# B&R Automation Studio project DevProj
Automation Studio 4.10.2.37; technology packages: mappMotion 5.12.3

## Configuration Config1

CPU 5APC2200.AL14-000, AutomationRuntime B4.91, Build 4.1.2, Safety 0.0, Vc V4.72.3

### Task classes (Cpu.sw)
```
Cyclic#1:
  Main <- Programs.Main.prg
Binaries: udbdef, FWRules, TCData, sysconf, Role, User, iomap, ashwd, asfw, arconfig, ashwac
Libraries: standard, operator, runtime, astime, AsIecCon, Util, McBase, MpAxis, McAxis, MpBase, McAcpAx, PTP
```

### Hardware
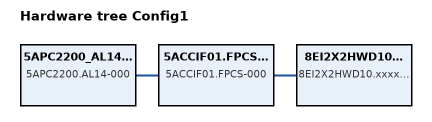
```
5ACCIF01.FPCS-000 : 5ACCIF01.FPCS-000 v1.8.1.0  [SL -> 5APC2200_AL14_000.SL1]
  Connector IF1:
    DNAConfiguration = manual
5APC2200_AL14_000 : 5APC2200.AL14-000 v2.0.1.0
  Connector IF3:
    AssignedOperatingSystem = ARemb
    ActivateDevice = 1
  Connector IF4:
    AssignedOperatingSystem = ARemb
    ActivateDevice = 1
  Connector IF5:
    AssignedOperatingSystem = ARemb
  Connector IF6:
    AssignedOperatingSystem = ARemb
  ConfigurationID = DevProj_Config1
  UserPartitionSize = 0
  TimerDeviceType = EPLX2X
  TimerDevice = 5ACCIF01.FPCS-000.IF1
  TaskClassIdleTime = 2000
  Cyclic1Tolerance = 0
  Cyclic2Duration = 10000
  Cyclic2Tolerance = 10000
  FileDevice1
  FileDeviceName1 = CNC_PrgDir
  FileDevicePath1 = C:\scUserFiles\
  ActivateOpcUa = 1
  OpcUa_AuthenticationSecurityPolicy_EnableNone = 1
  OpcUa_AuthenticationSecurityPolicy_EnableBasic128Rsa15 = 1
  OpcUa_Security_AdminRole = Everyone
  OpcUaLimitsMaxSessions = 4
  OpcUa_SamplingTimer_Default = 4
  OpcUaInformationModels_PV_Version = 1
8EI2X2HWD10.xxxx-1 : 8EI2X2HWD10.xxxx-1 v2.3.1.1  [PLK1 -> 5ACCIF01.FPCS-000.IF1 [Cable Type=PowerlinkCable, Length=10, Version=1.0.0.3]]
  DriveConfiguration/Module:
    McAcoposTypeID = AcoposP3DConfig
    ActivateACOPOSSimulationOnPLC = 1
  DriveConfiguration/Channel[1]/RealAxis:
    AxisReference = AxisX1_Link
  DriveConfiguration/Channel[1]/RealAxis/MechanicalElements/Gearbox:
    InputIsReadOnly = 0
    Input = 1
    OutputIsReadOnly = 0
    Output = 1
  DriveConfiguration/Channel[1]/RealAxis/MechanicalElements/RotaryToLinearTransformation:
    ReferenceDistanceIsReadOnly = 0
    ReferenceDistance = 1
  DriveConfiguration/Channel[1]/RealAxis/Controller:
    ModeIsReadOnly = 0
    Mode = PositionController
  DriveConfiguration/Channel[1]/RealAxis/Controller/Mode/Position:
    ProportionalGain = 50.0
    IntegrationTime = 0.0
    PredictionTime = 0.0004
    TotalDelayTime = 0.0004
  DriveConfiguration/Channel[1]/RealAxis/Controller/Mode/Speed:
    ProportionalGainIsReadOnly = 0
    ProportionalGain = 2.0
    IntegrationTimeIsReadOnly = 0
    IntegrationTime = 0.0
    FilterTimeIsReadOnly = 0
    FilterTime = 0.0
  DriveConfiguration/Channel[1]/RealAxis/Controller/Mode/LoopFilters:
    LoopFilter1 = NotUsed
    LoopFilter2 = NotUsed
    LoopFilter3 = NotUsed
  DriveConfiguration/Channel[1]/RealAxis/Homing:
    Mode = Direct
  DriveConfiguration/Channel[1]/RealAxis/Homing/Mode:
    Position = 0.0
    ReferencePulse = NotUsed
  DriveConfiguration/Channel[1]/RealAxis/Homing:
    RestorePositionVariable = 
  DriveConfiguration/Channel[1]/RealAxis/StopReaction:
    Quickstop = DecelerationLimit
    DriveError = DecelerationLimit
  DriveConfiguration/Channel[1]/RealAxis/MovementErrorLimits:
    PositionError = 1.0
    VelocityErrorMonitoring = Automatic1
  DriveConfiguration/Channel[1]/RealAxis:
    JerkFilter = NotUsed
  DriveConfiguration/Channel[1]/RealAxis/DigitalInputs/HomingSwitch:
    Source = NotUsed
    Level = High
  DriveConfiguration/Channel[1]/RealAxis/DigitalInputs/PositiveLimitSwitch:
    Source = NotUsed
    Level = High
  DriveConfiguration/Channel[1]/RealAxis/DigitalInputs/NegativeLimitSwitch:
    Source = NotUsed
    Level = High
  DriveConfiguration/Channel[1]/RealAxis/DigitalInputs/Trigger1:
    Source = X8Trigger1
    Level = High
  DriveConfiguration/Channel[1]/RealAxis/DigitalInputs/Trigger2:
    Source = X8Trigger2
    Level = High
  DriveConfiguration/Channel[1]/RealAxis/DigitalInputs/Quickstop:
    Input = Trigger2
  DriveConfiguration/Channel[1]/RealAxis/Simulation:
    SimulationModeOnPLC = SetValueGeneration
    SimulationModeOnACOPOS = NotUsed
  DriveConfiguration/Channel[2]/RealAxis:
    AxisReference = AxisZ1_Link
  DriveConfiguration/Channel[2]/RealAxis/MechanicalElements/Gearbox:
    InputIsReadOnly = 0
    Input = 1
    OutputIsReadOnly = 0
    Output = 1
  DriveConfiguration/Channel[2]/RealAxis/MechanicalElements/RotaryToLinearTransformation:
    ReferenceDistanceIsReadOnly = 0
    ReferenceDistance = 1
  DriveConfiguration/Channel[2]/RealAxis/Controller:
    ModeIsReadOnly = 0
    Mode = PositionController
  DriveConfiguration/Channel[2]/RealAxis/Controller/Mode/Position:
    ProportionalGain = 50.0
    IntegrationTime = 0.0
    PredictionTime = 0.0004
    TotalDelayTime = 0.0004
  DriveConfiguration/Channel[2]/RealAxis/Controller/Mode/Speed:
    ProportionalGainIsReadOnly = 0
    ProportionalGain = 2.0
    IntegrationTimeIsReadOnly = 0
    IntegrationTime = 0.0
    FilterTimeIsReadOnly = 0
    FilterTime = 0.0
  DriveConfiguration/Channel[2]/RealAxis/Controller/Mode/LoopFilters:
    LoopFilter1 = NotUsed
    LoopFilter2 = NotUsed
    LoopFilter3 = NotUsed
  DriveConfiguration/Channel[2]/RealAxis/Homing:
    Mode = Direct
  DriveConfiguration/Channel[2]/RealAxis/Homing/Mode:
    Position = 0.0
    ReferencePulse = NotUsed
  DriveConfiguration/Channel[2]/RealAxis/Homing:
    RestorePositionVariable = 
  DriveConfiguration/Channel[2]/RealAxis/StopReaction:
    Quickstop = DecelerationLimit
    DriveError = DecelerationLimit
  DriveConfiguration/Channel[2]/RealAxis/MovementErrorLimits:
    PositionError = 1.0
    VelocityErrorMonitoring = Automatic1
  DriveConfiguration/Channel[2]/RealAxis:
    JerkFilter = NotUsed
  DriveConfiguration/Channel[2]/RealAxis/DigitalInputs/HomingSwitch:
    Source = NotUsed
    Level = High
  DriveConfiguration/Channel[2]/RealAxis/DigitalInputs/PositiveLimitSwitch:
    Source = NotUsed
    Level = High
  DriveConfiguration/Channel[2]/RealAxis/DigitalInputs/NegativeLimitSwitch:
    Source = NotUsed
    Level = High
  DriveConfiguration/Channel[2]/RealAxis/DigitalInputs/Trigger1:
    Source = X8Trigger1
    Level = High
  DriveConfiguration/Channel[2]/RealAxis/DigitalInputs/Trigger2:
    Source = X8Trigger2
    Level = High
  DriveConfiguration/Channel[2]/RealAxis/DigitalInputs/Quickstop:
    Input = Trigger2
  DriveConfiguration/Channel[2]/RealAxis/Simulation:
    SimulationModeOnPLC = SetValueGeneration
    SimulationModeOnACOPOS = NotUsed
```

### ConfAxFea.axesgroupfeature - 5APC2200_AL14_000/mappMotion/ConfAxFea.axesgroupfeature
```
Element Feature_Programs (Type=axesgroupfeature)
  Type = Program
    ModalDataBehaviour = UseAxesGroupSettings
    InitialSettings:
      InterpolationTypes = LinearRapid
      PositionCoordinates = Absolute
      CircleCoordinates = Relative
      JACS_ACSProgramming = JACS
      ContourConnection = Inactive
      ProgrammingUnits = UseAxesGroupSettings
      Feedrates:
        FeedPath = Standard
        FeedCharacteristic = StandardCharacteristic
        FeedType = Feedrate
        FeedReduction = Inactive
        FeedrateValue = 0.0
        InverseFeedrateValue = 0.0
        FeedratePerRevValue = 0.0
    DefaultLanguage = BRGCode
    Location = Default
      FileDevice = CNC_PrgDir
    ProgramElements:
      PVs:
        PV[1]:
          PvName = ::RParams[31]
          Advanced:
            Alias = R31
            Synchronization = Ip
            Reference = No
Element Feature_Jogging (Type=axesgroupfeature)
  Type = Jogging
Element Feature_MFunctions (Type=axesgroupfeature)
  Type = MFunctions
    ModalDataBehaviour = UseAxesGroupSettings
    MFunction[1]:
      IndexType = Single
        Index = 31
      Blocking = Disabled
      Output = Before
      InSimulation = NotUsed
      PvMapping = ::M31
      Counter
```

### ConfAxes.axis - 5APC2200_AL14_000/mappMotion/ConfAxes.axis
```
Element AxisX1_Link (Type=axis)
  BaseTypeIsReadOnly = 0
  BaseType = LinearBounded
    MeasurementUnit = 5066068
    MeasurementResolutionIsReadOnly = 0
    MeasurementResolution = 0.01
    CountDirectionIsReadOnly = 0
    CountDirection = Standard
  MovementLimitsIsReadOnly = 0
  MovementLimits = Internal
    Position:
      LowerLimitMin = -1.79769313486231E308
      UpperLimitMax = 1.79769313486231E308
      LowerLimit = -1000.0
      UpperLimit = 1000.0
    VelocityIsReadOnly = 0
    Velocity:
      VelocityMax = 3.4E38
      Velocity = 10.0
    AccelerationIsReadOnly = 0
    Acceleration:
      AccelerationMax = 3.4E38
      Acceleration = 50.0
    DecelerationIsReadOnly = 0
    Deceleration:
      DecelerationMax = 3.4E38
      Deceleration = 50.0
  Alarms = None
Element AxisZ1_Link (Type=axis)
  BaseTypeIsReadOnly = 0
  BaseType = LinearBounded
    MeasurementUnit = 5066068
    MeasurementResolutionIsReadOnly = 0
    MeasurementResolution = 0.01
    CountDirectionIsReadOnly = 0
    CountDirection = Standard
  MovementLimitsIsReadOnly = 0
  MovementLimits = Internal
    Position:
      LowerLimitMin = -1.79769313486231E308
      UpperLimitMax = 1.79769313486231E308
      LowerLimit = -1000.0
      UpperLimit = 1000.0
    VelocityIsReadOnly = 0
    Velocity:
      VelocityMax = 3.4E38
      Velocity = 10.0
    AccelerationIsReadOnly = 0
    Acceleration:
      AccelerationMax = 3.4E38
      Acceleration = 50.0
    DecelerationIsReadOnly = 0
    Deceleration:
      DecelerationMax = 3.4E38
      Deceleration = 50.0
  Alarms = None
```

### ConfCnc.axesgroup - 5APC2200_AL14_000/mappMotion/ConfCnc.axesgroup
```
Element CncXZ_Link (Type=axesgroup)
  Type = PathGenAxesGroup
    ProcessingTaskClass = 1
    License = 1
    PhysicalAxes:
      JointAxes:
        JointAxis[1]:
          Name = QX
          AxisRef = AxisX1_Link
        JointAxis[2]:
          Name = QZ
          AxisRef = AxisZ1_Link
    MechanicalSystem:
      MechSysRef = MechSys_2AxCNCXZ
    BasicSettings:
      ModalDataBehaviour = ResetToDefault
      GeometryPlanning:
        RoundingMode = Standard
        MaxCornerDeviation = 0.0
        MaxTangentialTransitionDeviation = 0.0
        MaxRadiusDeviation = 0.001
        WorkingPlane = ZX
      TrajectoryPlanning = Basic
        LimitCheckResolution = UserDefinedTime
          Time = 0.01
        BufferTime = UserDefinedTime
          Time = 0.1
    AxesGroupFeatures:
      FeatureRef[1] = Feature_Programs
      FeatureRef[2] = Feature_Jogging
      FeatureRef[3] = Feature_MFunctions
  Alarms = None
```

### ConfigAx1.axis - 5APC2200_AL14_000/mappMotion/ConfigAx1.axis
```
Element AxisX1_Link (Type=axis)
  BaseTypeIsReadOnly = 0
  BaseType = LinearBounded
    MeasurementUnit = 5066068
    MeasurementResolutionIsReadOnly = 0
    MeasurementResolution = 0.01
    CountDirectionIsReadOnly = 0
    CountDirection = Standard
  MovementLimitsIsReadOnly = 0
  MovementLimits = Internal
    Position:
      LowerLimitMin = -1.79769313486231E308
      UpperLimitMax = 1.79769313486231E308
      LowerLimit = -1000.0
      UpperLimit = 1000.0
    VelocityIsReadOnly = 0
    Velocity:
      VelocityMax = 3.4E38
      Velocity = 10.0
    AccelerationIsReadOnly = 0
    Acceleration:
      AccelerationMax = 3.4E38
      Acceleration = 50.0
    DecelerationIsReadOnly = 0
    Deceleration:
      DecelerationMax = 3.4E38
      Deceleration = 50.0
  Alarms = MpAlarmX
```

### ConfigAx2.axis - 5APC2200_AL14_000/mappMotion/ConfigAx2.axis
```
Element AxisZ1_Ref (Type=axis)
  BaseTypeIsReadOnly = 0
  BaseType = LinearBounded
    MeasurementUnit = 5066068
    MeasurementResolutionIsReadOnly = 0
    MeasurementResolution = 0.01
    CountDirectionIsReadOnly = 0
    CountDirection = Standard
  MovementLimitsIsReadOnly = 0
  MovementLimits = Internal
    Position:
      LowerLimitMin = -1.79769313486231E308
      UpperLimitMax = 1.79769313486231E308
      LowerLimit = -1000.0
      UpperLimit = 1000.0
    VelocityIsReadOnly = 0
    Velocity:
      VelocityMax = 3.4E38
      Velocity = 10.0
    AccelerationIsReadOnly = 0
    Acceleration:
      AccelerationMax = 3.4E38
      Acceleration = 50.0
    DecelerationIsReadOnly = 0
    Deceleration:
      DecelerationMax = 3.4E38
      Deceleration = 50.0
  Alarms = None
```

### Config_1.axesgroupfeature - 5APC2200_AL14_000/mappMotion/Config_1.axesgroupfeature
```
Element Feature_MFunctions (Type=axesgroupfeature)
  Type = MFunctions
    ModalDataBehaviour = UseAxesGroupSettings
    MFunction[1]:
      IndexType = Range
        IndexTo = 100
      Blocking = Enabled
      Output = Before
      InSimulation = Set
      PvMapping = ::MFunc
      Counter
```

## Logical view

Binary libraries used (declarations not repeated): operator, runtime, astime, AsIecCon, standard, McBase 5.13.2, McAcpAx 5.13.2, McAxis 5.13.2, MpAxis 5.13.2, MpBase 5.13.0, McBase 5.12.3, McAcpAx 5.12.3, McPathGen 5.12.3, McAxGroup 5.12.3, McAxis 5.12.3, McProgInt 5.12.3, MpCnc 5.12.3, MpAxis 5.12.3, MpBase

### Global.typ - Global data types
```iecst
TYPE
	T_HmiAxis : 	STRUCT
		Enabled : BOOL;
		ActPos : LREAL;
		Reset : BOOL;
		JogPlus : BOOL;
		JogMinus : BOOL;
		JogVelo : REAL;
		MoveSetPos : BOOL;
		SetVelo : REAL;
		SetPos : LREAL;
	END_STRUCT;
	T_Hmi : 	STRUCT
		StartMachine : BOOL;
		Axis : ARRAY[0..C_AXIS_COUNT]OF T_HmiAxis;
	END_STRUCT;
END_TYPE
```

### Global.var - Global variables
```iecst
VAR
	AxisX1 : T_Axis;
	AxisZ1 : T_Axis;
	CncChInfo : MpCnc2AxisInfoType;
	CncChParams : MpCnc2AxisParType;
	count : USINT;
	fbAxCtrlX1 : FB_AxisControl;
	fbAxCtrlZ1 : FB_AxisControl;
	fbCncChannel : MpCnc2Axis;
	HMI : T_Hmi;
	RParams : ARRAY[0..200] OF LREAL := [31(0.0),35,169(0.0)];
	M31 : BOOL;
	BRPlcVar2 : LREAL;
	BRPlcVar1 : UINT;
	Alarm : ARRAY[0..200] OF BOOL;
	strvar1 : STRING[80];
END_VAR
```

### GlobalConstant.var
```iecst
VAR CONSTANT
	C_AXIS_COUNT : USINT := 3;
END_VAR
```

### Package Logical/Libraries - Global libraries

### Library Logical/Libraries/_Haffner/PTP (IEC)

#### Types.typ - Exported data types
```iecst
TYPE
	T_AxisInterface : 	STRUCT
		IN : T_AxisInterfaceIn;
		OUT : T_AxisInterfaceOut;
	END_STRUCT;
	T_AxisInterfaceIn : 	STRUCT
		Enable : BOOL;
		Power : BOOL;
		Interlock : BOOL;
		Reset : BOOL;
		SetActPosVal : LREAL; (* Setlenecek pozisyon degeri *)
		SetActPos : BOOL;
		DriveReset : BOOL;
		MoveSetPos : BOOL;
		Home : BOOL;
		HomeSensor : BOOL;
		JogFw : BOOL;
		JogBw : BOOL;
		ReadDiagMsg : BOOL;
		HomePos : LREAL;
		SetPos : LREAL;
		SetVelo : REAL;
		SetAcc : LREAL;
		SetDec : LREAL;
		SetJerk : LREAL;
		JogVelo : REAL;
		Couple : BOOL;
		CoupleRef : REFERENCE TO McAxisType;
		Override : LREAL := 100.0;
	END_STRUCT;
	T_AxisInterfaceOut : 	STRUCT
		Enabled : BOOL;
		Powered : BOOL;
		Homed : BOOL;
		MoveDone : BOOL;
		DiagMsgError : BOOL;
		DiagMessage : STRING[80];
		ErrID : DINT;
		Error : BOOL;
	END_STRUCT;
	T_AxisParams : 	STRUCT
		WriteParam : BOOL;
		Calibrate : BOOL;
		WritePositionBias : BOOL;
		WriteParamDone : BOOL;
		CalibrationDone : BOOL;
		CalcPositionBias : LREAL;
		Error : BOOL;
		ErrorId : UDINT;
		PositionBias : LREAL;
		MinLimitPos : LREAL;
		MaxLimitPos : LREAL;
		HomePos : LREAL;
		GroundPos : LREAL;
		MaxVelo : LREAL;
		RapidTraverseVelo : LREAL;
		MoveVelo : LREAL;
		MinLimitEnabled : BOOL;
		MaxLimitEnabled : BOOL;
		CalibrationPos : LREAL;
		PositionTolerance : LREAL;
		RefStatus : LREAL; (* 0: Not referenced, 1: Referenced, 2: Homing axis *)
	END_STRUCT;
	T_Axis : 	STRUCT
		Ctrl : T_AxisInterface;
		Params : T_AxisParams;
		ID : UINT;
		AbsEnc : BOOL;
		Installed : BOOL;
		Ref : T_AxisRef;
	END_STRUCT;
	T_AxisRef : 	STRUCT
		ActPos : LREAL;
	END_STRUCT;
END_TYPE
```

#### PTP.fun - Exported functions and function blocks
```iecst
FUNCTION_BLOCK FB_AxisControl
	VAR_IN_OUT
		stAxisInterface : T_AxisInterface;
		stAxisParams : T_AxisParams;
		AxisLink : McAxisType;
	END_VAR
	VAR
		fbMpAxisBasic : MpAxisBasic;
		tMpAxisBasicParType : MpAxisBasicParType;
	END_VAR
	VAR_IN_OUT
		AxisRef : T_AxisRef;
	END_VAR
END_FUNCTION_BLOCK
```

#### FB_AxisControl.st
```iecst
FUNCTION_BLOCK FB_AxisControl

	tMpAxisBasicParType.Position			:= stAxisInterface.IN.SetPos;
	tMpAxisBasicParType.Velocity			:= stAxisInterface.IN.SetVelo;
	tMpAxisBasicParType.Jog.Velocity		:= stAxisInterface.IN.JogVelo;

	IF stAxisParams.Calibrate THEN
		tMpAxisBasicParType.Homing.Position	:= stAxisParams.CalibrationPos;
		tMpAxisBasicParType.Homing.Mode		:= mcHOMING_DIRECT;
		fbMpAxisBasic.Home					:= TRUE;
		stAxisParams.CalibrationDone		:= fbMpAxisBasic.IsHomed;

	ELSIF stAxisParams.WritePositionBias THEN
		tMpAxisBasicParType.Homing.Mode		:= mcHOMING_ABSOLUTE;
		fbMpAxisBasic.Home					:= TRUE;
		stAxisParams.WriteParamDone			:= fbMpAxisBasic.IsHomed;

	ELSE
		fbMpAxisBasic.Home					:= FALSE;
	END_IF

	IF NOT stAxisParams.Calibrate THEN
		stAxisParams.CalibrationDone		:= FALSE;
	END_IF

	IF NOT stAxisParams.WritePositionBias AND NOT stAxisParams.WriteParam THEN
		stAxisParams.WriteParamDone			:= FALSE;
	END_IF

	fbMpAxisBasic(
		MpLink			:= ADR(AxisLink),
		Enable			:= stAxisInterface.IN.Enable,
		ErrorReset		:= stAxisInterface.IN.Reset,
		Parameters		:= ADR(tMpAxisBasicParType),
		(*		Update			:=, 	*)
		Power			:=  fbMpAxisBasic.Info.ReadyToPowerOn AND stAxisInterface.IN.Power,
		(*		Home			:= stAxisInterface.IN.Home,	*)
		(*		MoveVelocity	:= ,	*)
		MoveAbsolute	:= stAxisInterface.IN.MoveSetPos,
		(*		MoveAdditive	:= , *)
		(*		Stop			:= , *)
		JogPositive		:= stAxisInterface.IN.JogFw,
		JogNegative		:= stAxisInterface.IN.JogBw,
		(*		LimitLoad		:= ,	ReleaseBrake	:= ,*)
		);

	stAxisInterface.OUT.Enabled		:= fbMpAxisBasic.Active;
	stAxisInterface.OUT.Error		:= fbMpAxisBasic.Error;
	stAxisInterface.OUT.ErrID		:= fbMpAxisBasic.StatusID;
	stAxisInterface.OUT.Powered		:= fbMpAxisBasic.PowerOn;
	stAxisInterface.OUT.MoveDone	:= fbMpAxisBasic.MoveDone;
	stAxisInterface.OUT.Homed		:= fbMpAxisBasic.IsHomed;
	AxisRef.ActPos					:= fbMpAxisBasic.Position;

END_FUNCTION_BLOCK
```

### Library Logical/Libraries/_Haffner/Util (IEC)

#### Types.typ - Exported data types
```iecst
TYPE
	E_CylinderModes :
		(
		_tbsg := 0, (* tek bobin, sensor geride				*)
		_tbsi := 1, (* tek bobin, sensor ileride				*)
		_tbcs := 2, (* tek bobin, cift sensor					*)
		_cbsg := 3, (* cift bobin, sensor geride				*)
		_cbsi := 4, (* cift bobin, sensor ileride				*)
		_cbcs := 5, (* cift bobin cift sensor					*)
		_tbsy := 6, (* tek bobin, sensor yok					*)
		_cbsy := 7, (* cift bobin, sensor yok					*)
		_casy := 8, (* cift bobin acik merkez, sensor yok		*)
		_casg := 10 (* cift bobin acik merkez, sensor geride	*)
		);
END_TYPE
```

#### Util.fun - Exported functions and function blocks
```iecst
FUNCTION_BLOCK FB_CylinderControl
	VAR_INPUT
		Emergency : BOOL;
		Enabled : BOOL;
		Mode : E_CylinderModes;
		OnRstPosSensor : BOOL;
		OnRstPosTime : UINT;
		OnSetPosSensor : BOOL;
		OnSetPosTime : UINT;
		AlarmTime : UINT;
		AlarmAck : BOOL;
		ID : UINT;
		Simulation : BOOL;
		Rst : BOOL;
		Set : BOOL;
	END_VAR
	VAR_OUTPUT
		OutRst : BOOL;
		OutSet : BOOL;
		OnRstPos : BOOL;
		OnSetPos : BOOL;
		OutRstAlm : BOOL;
		OutSetAlm : BOOL;
	END_VAR
	VAR
		tonSet : TON;
		tonRst : TON;
		rtSet : R_TRIG;
		ftSet : F_TRIG;
		rtRst : R_TRIG;
		ftRst : F_TRIG;
		FilterTime : TIME := T#50ms;
		NoSetSensor : BOOL;
		NoRstSensor : BOOL;
		SingleActing : BOOL;
		DoubleActing : BOOL;
		StateRst : UINT;
		StateSet : UINT;
		tonSetAlarm : TON;
		tonRstAlarm : TON;
		OpenCenter : BOOL;
		rtActCmd : R_TRIG;
		actCmd : UINT;
		prevCmd : UINT;
		ftEmergency : F_TRIG;
	END_VAR
END_FUNCTION_BLOCK
```

#### FB_CylinderControl.st
```iecst
FUNCTION_BLOCK FB_CylinderControl

	(*****************************************************************************************************************************)
	rtRst(CLK := Rst AND Enabled AND NOT Emergency);
	ftRst(CLK := Rst AND Enabled AND NOT Emergency);

	rtSet(CLK := Set AND Enabled AND NOT Emergency);
	ftSet(CLK := Set AND Enabled AND NOT Emergency);

	IF rtSet.Q THEN	actCmd := 2;	END_IF
	IF rtRst.Q THEN	actCmd := 1;	END_IF
	rtActCmd(CLK := actCmd <> prevCmd);
	prevCmd				:= actCmd;

	NoRstSensor			:= Mode = _tbsi OR Mode = _cbsi OR Mode = _tbsy OR Mode = _cbsy OR Mode = _casy;
	NoSetSensor			:= Mode = _tbsg OR Mode = _cbsg OR Mode = _tbsy OR Mode = _cbsy OR Mode = _casy;
	SingleActing		:= Mode = _tbsg OR Mode = _tbsi OR Mode = _tbcs OR Mode = _tbsy;
	DoubleActing		:= Mode = _cbsg OR Mode = _cbsi OR Mode = _cbcs OR Mode = _cbsy OR Mode = _casy;
	OpenCenter			:= Mode = _casy OR Mode = _casg;
	(*****************************************************************************************************************************)
	CASE StateRst OF
		0:
			tonRst(IN := FALSE);

			tonRstAlarm.IN		:= FALSE;
			OutRst				:= FALSE;
			OnRstPos			:= FALSE;
			OutRstAlm			:= FALSE;

		10:
			Set					:= FALSE;
			StateSet				:= 0;
			StateRst				:= 20;

		20:
			OutRst				:= NOT Simulation;

			IF Simulation THEN
				tonRst.IN			:= TRUE;
				tonRst.PT			:=  UINT_TO_TIME(OnRstPosTime);
				tonRstAlarm.IN	:= FALSE;
				tonRstAlarm.PT	:= UINT_TO_TIME(AlarmTime);

			ELSIF NOT NoRstSensor THEN											(* Reset pos sensoru varsa *)
				tonRst.IN			:= OnRstPosSensor;
				tonRst.PT			:= FilterTime;
				tonRstAlarm.IN	:= NOT OnRstPosSensor;
				tonRstAlarm.PT	:= UINT_TO_TIME(AlarmTime);

			ELSIF NOT NoSetSensor THEN											(* Reset pos sensoru yok, Set pos sensoru varsa *)
				tonRst.IN			:= NOT OnSetPosSensor;
				tonRst.PT			:= UINT_TO_TIME(OnRstPosTime);
				tonRstAlarm.IN	:= OnSetPosSensor;
				tonRstAlarm.PT	:= UINT_TO_TIME(AlarmTime);

			ELSE
				tonRst.IN			:= TRUE;
				tonRst.PT			:= UINT_TO_TIME(OnRstPosTime);
				tonRstAlarm.IN	:= FALSE;
			END_IF

			tonRst();
			IF tonRst.Q AND NOT OutRstAlm THEN
				StateRst			:= 30;
			END_IF

		30:
			OutRst				:= NOT Simulation AND (NOT OpenCenter AND (SingleActing OR DoubleActing) OR (OpenCenter AND Rst));
			OnRstPos			:= (NOT OpenCenter AND (SingleActing OR DoubleActing) OR (OpenCenter AND Rst));
	END_CASE
	(*****************************************************************************************************************************)
	tonRstAlarm();
	IF tonRstAlarm.Q THEN
		OutRstAlm		:= TRUE;
	ELSIF AlarmAck THEN
		OutRstAlm		:= FALSE;
	END_IF
	(*****************************************************************************************************************************)
	CASE StateSet OF
		0:
			tonSet(IN := FALSE);

			tonSetAlarm.IN		:= FALSE;
			OutSet				:= FALSE;
			OnSetPos			:= FALSE;
			OutSetAlm			:= FALSE;

		10:
			Rst					:= FALSE;
			StateRst				:= 0;
			StateSet				:= 20;

		20:
			OutSet				:= NOT Simulation;

			IF Simulation THEN
				tonSet.IN			:= TRUE;
				tonSet.PT			:=  UINT_TO_TIME(OnRstPosTime);
				tonSetAlarm.IN	:= FALSE;
				tonSetAlarm.PT	:= UINT_TO_TIME(AlarmTime);

			ELSIF NOT NoSetSensor THEN
				tonSet.IN			:= OnSetPosSensor;
				tonSet.PT			:= FilterTime;
				tonSetAlarm.IN	:= NOT OnSetPosSensor;
				tonSetAlarm.PT	:= UINT_TO_TIME(AlarmTime);

			ELSIF NOT NoRstSensor THEN
				tonSet.IN			:= NOT OnRstPosSensor;
				tonSet.PT			:= UINT_TO_TIME(OnSetPosTime);
				tonSetAlarm.IN	:= OnRstPosSensor;
				tonSetAlarm.PT	:= UINT_TO_TIME(AlarmTime);

			ELSE
				tonSet.IN			:= NOT tonSetAlarm.Q;
				tonSet.PT			:= UINT_TO_TIME(OnSetPosTime);
				tonSetAlarm.IN	:= FALSE;
			END_IF

			tonSet();

			IF tonSet.Q AND NOT OutSetAlm THEN
				StateSet			:= 30;
			END_IF

		30:
			OutSet				:= NOT Simulation AND (NOT OpenCenter AND (SingleActing OR DoubleActing) OR (OpenCenter AND Set));
			OnSetPos			:= (NOT OpenCenter AND (SingleActing OR DoubleActing) OR (OpenCenter AND Set));
	END_CASE
	(*****************************************************************************************************************************)
	tonSetAlarm();
	IF tonSetAlarm.Q THEN
		OutSetAlm			:= TRUE;
	ELSIF AlarmAck THEN
		OutSetAlm			:= FALSE;
	END_IF
	(*****************************************************************************************************************************)
	IF Emergency OR NOT Enabled THEN
		StateRst				:= 0;
		StateSet				:= 0;
	END_IF

	ftEmergency(CLK := Emergency);
	IF NOT Enabled THEN
		OutRstAlm			:=
		OutSetAlm			:= FALSE;
		OnRstPos			:=
		OnSetPos			:= TRUE;

	ELSIF Emergency THEN
		OutRstAlm			:=
		OutSetAlm			:= FALSE;

	ELSIF ftEmergency.Q THEN
		IF actCmd = 2 THEN
			StateSet			:= 30;
		ELSE
			StateRst			:= 30;
		END_IF

	ELSE
		IF rtRst.Q OR (Rst AND ftSet.Q) THEN
			OnSetPos		:=
			Set				:= FALSE;
			StateSet			:= 0;
			IF NOT OnRstPos THEN
				StateRst		:= 10;
			END_IF
		END_IF

		IF rtSet.Q OR (Set AND ftRst.Q) THEN
			OnRstPos		:=
			Rst				:= FALSE;
			StateRst			:= 0;
			IF NOT OnSetPos THEN
				StateSet		:= 10;
			END_IF
		END_IF
	END_IF

END_FUNCTION_BLOCK
```

### Program Logical/Programs/PRG_Main (IEC)

#### Variables.var
```iecst
VAR
	fbCyCo1 : FB_CylinderControl;
END_VAR
```

#### Main.st
```iecst
PROGRAM _INIT
	(* Insert code here *)

END_PROGRAM

PROGRAM _CYCLIC

	fbCyCo1(
		Emergency := FALSE,
		Enabled := TRUE,
		Mode := _tbsy,
		OnRstPosSensor := FALSE,
		OnRstPosTime := 1000,
		OnSetPosSensor := FALSE,
		OnSetPosTime := 1000,
		AlarmTime := 2000,
		AlarmAck := FALSE,
		ID := 1,
		Simulation := FALSE,
//		Rst :=
//		Set :=
		);

//Hmi and plc assigning
//AxisX1
	HMI.Axis[0].Enabled			:= AxisX1.Ctrl.OUT.Powered;
	HMI.Axis[0].ActPos			:= AxisX1.Ref.ActPos;

	AxisX1.Ctrl.IN.Reset		:= HMI.Axis[0].Reset;
	AxisX1.Ctrl.IN.JogVelo		:= HMI.Axis[0].JogVelo;
	AxisX1.Ctrl.IN.JogFw		:= HMI.Axis[0].JogPlus;
	AxisX1.Ctrl.IN.JogBw		:= HMI.Axis[0].JogMinus;

	AxisX1.Ctrl.IN.MoveSetPos	:= HMI.Axis[0].MoveSetPos;
	AxisX1.Ctrl.IN.SetVelo		:= HMI.Axis[0].SetVelo;
	AxisX1.Ctrl.IN.SetPos		:= HMI.Axis[0].SetPos;

//AxisZ1
	HMI.Axis[1].Enabled			:= AxisZ1.Ctrl.OUT.Powered;
	HMI.Axis[1].ActPos			:= AxisZ1.Ref.ActPos;

	AxisZ1.Ctrl.IN.Reset		:= HMI.Axis[1].Reset;
	AxisZ1.Ctrl.IN.JogVelo		:= HMI.Axis[1].JogVelo;
	AxisZ1.Ctrl.IN.JogFw		:= HMI.Axis[1].JogPlus;
	AxisZ1.Ctrl.IN.JogBw		:= HMI.Axis[1].JogMinus;

	AxisZ1.Ctrl.IN.MoveSetPos	:= HMI.Axis[1].MoveSetPos;
	AxisZ1.Ctrl.IN.SetVelo		:= HMI.Axis[1].SetVelo;
	AxisZ1.Ctrl.IN.SetPos		:= HMI.Axis[1].SetPos;

	BRPlcVar1;
	BRPlcVar2;
	Alarm;
	strvar1;

END_PROGRAM

PROGRAM _EXIT
	(* Insert code here *)

END_PROGRAM
```

### Program Logical/Programs/Sayici (IEC)

#### Main.st
```iecst
PROGRAM _INIT
	(* Insert code here *)

END_PROGRAM

PROGRAM _CYCLIC

	HMI.StartMachine := HMI.StartMachine;
	IF count < 200 THEN
		count := count + 1;
	ELSE
		count := 0;
	END_IF

END_PROGRAM

PROGRAM _EXIT
	(* Insert code here *)

END_PROGRAM
```

### Program Logical/Programs/PRG_Axes (IEC)

#### Variables.var
```iecst
VAR
	stateAxX1 : UINT;
END_VAR
```

#### Main.st
```iecst
PROGRAM _INIT
	(* Insert code here *)

END_PROGRAM

PROGRAM _CYCLIC

	CASE stateAxX1 OF
		0:
			stateAxX1	:= stateAxX1 + 10;

		10:
			AxisX1.Ctrl.IN.Enable			:= TRUE;
			AxisX1.Params.WriteParam		:= FALSE;

			AxisZ1.Ctrl.IN.Enable			:= TRUE;
			AxisZ1.Params.WriteParam		:= FALSE;

			IF AxisX1.Ctrl.OUT.Enabled AND NOT AxisX1.Params.WriteParamDone
			AND AxisZ1.Ctrl.OUT.Enabled AND NOT AxisZ1.Params.WriteParamDone THEN
				stateAxX1					:= stateAxX1 + 10;
			END_IF

		20:
			AxisX1.Params.WritePositionBias		:= TRUE;
			AxisZ1.Params.WritePositionBias		:= TRUE;

			IF AxisX1.Params.WriteParamDone AND AxisZ1.Params.WriteParamDone THEN
				AxisX1.Params.WritePositionBias	:= FALSE;
				AxisZ1.Params.WritePositionBias	:= FALSE;
				stateAxX1						:= stateAxX1 + 10;
			END_IF

			//			AxisX1.Ctrl.IN.HomePos	:= 100;
			//			AxisX1.Ctrl.IN.Home		:= TRUE;
			//
			//			IF AxisX1.Ctrl.OUT.Homed THEN
			//				AxisX1.Ctrl.IN.Home	:= FALSE;
			//				stateAxX1			:= stateAxX1 + 10;
			//			END_IF

		30:
			AxisX1.Ctrl.IN.JogVelo	:= 100;
			AxisX1.Ctrl.IN.Power	:= TRUE;

			AxisZ1.Ctrl.IN.JogVelo	:= 100;
			AxisZ1.Ctrl.IN.Power	:= TRUE;

			IF AxisX1.Ctrl.OUT.Powered AND AxisZ1.Ctrl.OUT.Powered THEN
				stateAxX1			:= stateAxX1 + 10;
			END_IF

		40:
			;

	END_CASE

	fbAxCtrlX1(
	stAxisInterface := AxisX1.Ctrl,
	stAxisParams 	:= AxisX1.Params,
	AxisLink 		:= AxisX1_Link,
	AxisRef			:= AxisX1.Ref
	);

	fbAxCtrlZ1(
	stAxisInterface := AxisZ1.Ctrl,
	stAxisParams 	:= AxisZ1.Params,
	AxisLink 		:= AxisZ1_Link,
	AxisRef			:= AxisZ1.Ref
	);

END_PROGRAM

PROGRAM _EXIT
	(* Insert code here *)

END_PROGRAM
```

### Program Logical/Programs/PRG_CNC (IEC)

#### Variables.var
```iecst
VAR
	State : UINT;
	fbBRMFunc : ARRAY[0..100] OF MC_BR_MFunction;
END_VAR
```

#### Main.st
```iecst
PROGRAM _INIT
	(* Insert code here *)
	M31;
	RParams;

	CncChParams.ProgramName := 'CncProg.cnc';

	fbCncChannel.MpLink				:= ADR(CncXZ_Link);
	fbCncChannel.Enable				:= TRUE;
	fbCncChannel.Override			:= 10;
	fbCncChannel.RapidOverride		:= 20;
	fbCncChannel.FeedrateOverride	:= 30;
	fbCncChannel.Parameters			:= ADR(CncChParams);

END_PROGRAM

PROGRAM _CYCLIC

	CASE State OF
		0:
			;
		10:
			IF AxisX1.Ctrl.OUT.Powered AND AxisX1.Ctrl.OUT.Homed
			AND AxisZ1.Ctrl.OUT.Powered AND AxisZ1.Ctrl.OUT.Homed THEN
				RParams[31]		:= 30;
				State			:= State + 10;
			END_IF

		20:
			IF fbCncChannel.Active THEN
				fbCncChannel.Power	:= TRUE;
			END_IF

			IF fbCncChannel.PowerOn THEN
				State				:= State + 10;
			END_IF

		30:
			fbCncChannel.MoveProgram	:= TRUE;

			IF fbCncChannel.MoveDone THEN
				State					:= State + 10;
			END_IF

		40:
			fbCncChannel.MoveProgram	:= FALSE;
			State						:= State + 10;

	END_CASE;

	fbCncChannel();

END_PROGRAM

PROGRAM _EXIT
	(* Insert code here *)

END_PROGRAM
```

### Program Logical/Programs/Main (IEC)

#### Main.st - Init, cyclic, exit code
```iecst
PROGRAM _INIT
	(* Insert code here *)

END_PROGRAM

PROGRAM _CYCLIC

	ACT_AxisX1;

	IF in1 THEN
		out1 := TRUE;
	ELSIF in2 THEN
		out1 := FALSE;
	END_IF

	fbCyCo1(
		Emergency := FALSE,
		Enabled := TRUE,
		Mode := _tbsy,
		OnRstPosSensor := FALSE,
		OnRstPosTime := 1000,
		OnSetPosSensor := FALSE,
		OnSetPosTime := 1000,
		AlarmTime := 2000,
		AlarmAck := FALSE,
		ID := 1,
		Simulation := FALSE,
//		Rst :=
//		Set :=
		);

END_PROGRAM

PROGRAM _EXIT
	(* Insert code here *)

END_PROGRAM
```

#### Variables.var - Local variables
```iecst
VAR
	in1 : BOOL;
	in2 : BOOL;
	out1 : BOOL;
	fbCyCo1 : FB_CylinderControl;
	fbAxCtrlX1 : FB_AxisControl;
	stateAxX1 : USINT;
END_VAR
```

#### ACT_AxisX1.st
```iecst
ACTION ACT_AxisX1:

	CASE stateAxX1 OF
		0:
			AxisX1.Ctrl.IN.Enable			:= TRUE;
			AxisX1.Params.WriteParam		:= FALSE;
			IF AxisX1.Ctrl.OUT.Enabled AND NOT AxisX1.Params.WriteParamDone THEN
				stateAxX1					:= stateAxX1 + 10;
			END_IF

		10:
			AxisX1.Params.WritePositionBias		:= TRUE;

			IF AxisX1.Params.WriteParamDone THEN
				AxisX1.Params.WritePositionBias	:= FALSE;
				stateAxX1						:= stateAxX1 + 10;
			END_IF

//			AxisX1.Ctrl.IN.HomePos	:= 100;
//			AxisX1.Ctrl.IN.Home		:= TRUE;
//
//			IF AxisX1.Ctrl.OUT.Homed THEN
//				AxisX1.Ctrl.IN.Home	:= FALSE;
//				stateAxX1			:= stateAxX1 + 10;
//			END_IF

		20:
			AxisX1.Ctrl.IN.JogVelo	:= 100;
			AxisX1.Ctrl.IN.Power	:= TRUE;
			IF AxisX1.Ctrl.OUT.Powered THEN
				stateAxX1			:= stateAxX1 + 10;
			END_IF

		30:
			;

	END_CASE

	fbAxCtrlX1
	(
		stAxisInterface := AxisX1.Ctrl,
		stAxisParams 	:= AxisX1.Params,
		AxisLink 		:= AxisX1_Link,
		AxisRef			:= AxisX1.Ref
	);

	HMI.Axis[0].Enabled	:= AxisX1.Ctrl.OUT.Powered;
	HMI.Axis[0].ActPos	:= AxisX1.Ref.ActPos;

	AxisX1.Ctrl.IN.Reset	:= HMI.Axis[0].Reset;
	AxisX1.Ctrl.IN.JogVelo	:= HMI.Axis[0].JogVelo;
	AxisX1.Ctrl.IN.JogFw	:= HMI.Axis[0].JogPlus;
	AxisX1.Ctrl.IN.JogBw	:= HMI.Axis[0].JogMinus;

	AxisX1.Ctrl.IN.MoveSetPos	:= HMI.Axis[0].MoveSetPos;
	AxisX1.Ctrl.IN.SetVelo		:= HMI.Axis[0].SetVelo;
	AxisX1.Ctrl.IN.SetPos		:= HMI.Axis[0].SetPos;

END_ACTION
```

- Visualisation Logical/Visu800x400 (not shown)

### Data object Logical/CncProg (Cnc)

#### CncProg.cnc - CNC program (G-Code)
```
%001 (CncProgram)

N10 G90
N20 F300
N30 G01 X30 Z30

N999 M30
```

Listed in the project but not available here: Logical/Libraries/_Haffner/PTP/Constants.var, Logical/Libraries/_Haffner/Util/Constants.var, Logical/Programs/Main/Types.typ
